(* LS Electric XG5000 project: hmi_연동 *)
(* PLC LSPLC *)

PROGRAM NewProgram (* task: 스캔 프로그램 *)

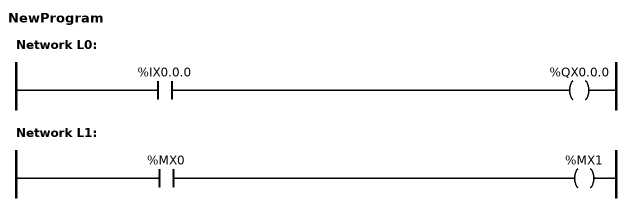
(* Rung L0 *)
%QX0.0.0 := %IX0.0.0;
(* Rung L1 *)
%MX1 := %MX0;
END_PROGRAM